// TIA Portal V19 export
FUNCTION "SET PARAMETER" : Void   // FC18, LAD
{ S7_Optimized_Access := 'TRUE' }
// stored: SetENOAutomatically false
   VAR_TEMP   // added for the SCL form of the ladder/FBD networks
      _w1 : Bool;
   END_VAR
BEGIN

REGION Network 1: MFG STIRRER MOTOR
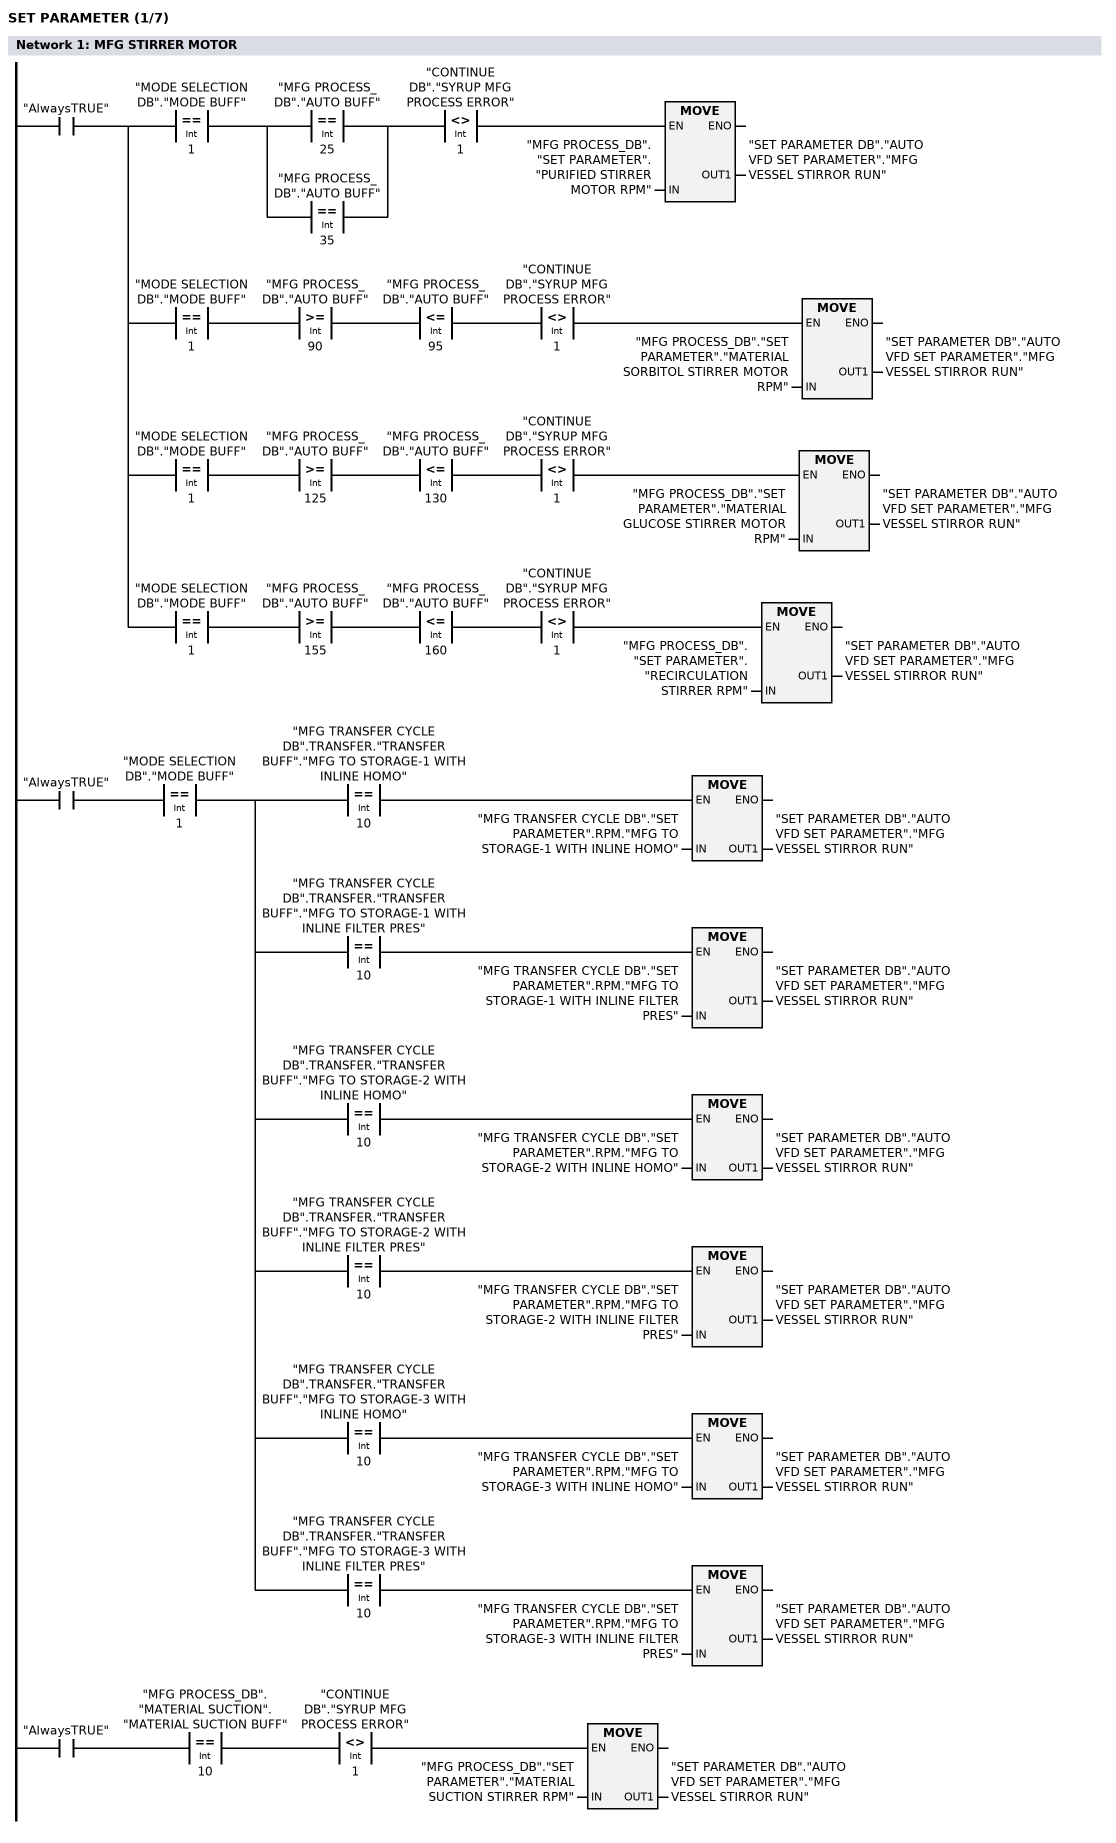
   RUNG wire#powerrail
      Contact( "AlwaysTRUE" )
      wire#w1
      { S7_Templates := "SrcType := Int" } EQ_Contact(in1 := "MODE SELECTION DB"."MODE BUFF", in2 := 1)
      wire#w2
      { S7_Templates := "SrcType := Int" } EQ_Contact(in1 := "MFG PROCESS_DB"."AUTO BUFF", in2 := 25)
      wire#w3
      { S7_Templates := "SrcType := Int" } NE_Contact(in1 := "CONTINUE DB"."SYRUP MFG PROCESS ERROR", in2 := 1)
      Move(in := "MFG PROCESS_DB"."SET PARAMETER"."PURIFIED STIRRER MOTOR RPM", out1 => "SET PARAMETER DB"."AUTO VFD SET PARAMETER"."MFG VESSEL STIRROR RUN")
   END_RUNG
   RUNG wire#w2
      { S7_Templates := "SrcType := Int" } EQ_Contact(in1 := "MFG PROCESS_DB"."AUTO BUFF", in2 := 35)
   END_RUNG wire#w3
   RUNG wire#w1
      { S7_Templates := "SrcType := Int" } EQ_Contact(in1 := "MODE SELECTION DB"."MODE BUFF", in2 := 1)
      { S7_Templates := "SrcType := Int" } GE_Contact(in1 := "MFG PROCESS_DB"."AUTO BUFF", in2 := 90)
      { S7_Templates := "SrcType := Int" } LE_Contact(in1 := "MFG PROCESS_DB"."AUTO BUFF", in2 := 95)
      { S7_Templates := "SrcType := Int" } NE_Contact(in1 := "CONTINUE DB"."SYRUP MFG PROCESS ERROR", in2 := 1)
      Move(in := "MFG PROCESS_DB"."SET PARAMETER"."MATERIAL SORBITOL STIRRER MOTOR RPM", out1 => "SET PARAMETER DB"."AUTO VFD SET PARAMETER"."MFG VESSEL STIRROR RUN")
   END_RUNG
   RUNG wire#w1
      { S7_Templates := "SrcType := Int" } EQ_Contact(in1 := "MODE SELECTION DB"."MODE BUFF", in2 := 1)
      { S7_Templates := "SrcType := Int" } GE_Contact(in1 := "MFG PROCESS_DB"."AUTO BUFF", in2 := 125)
      { S7_Templates := "SrcType := Int" } LE_Contact(in1 := "MFG PROCESS_DB"."AUTO BUFF", in2 := 130)
      { S7_Templates := "SrcType := Int" } NE_Contact(in1 := "CONTINUE DB"."SYRUP MFG PROCESS ERROR", in2 := 1)
      Move(in := "MFG PROCESS_DB"."SET PARAMETER"."MATERIAL GLUCOSE STIRRER MOTOR RPM", out1 => "SET PARAMETER DB"."AUTO VFD SET PARAMETER"."MFG VESSEL STIRROR RUN")
   END_RUNG
   RUNG wire#w1
      { S7_Templates := "SrcType := Int" } EQ_Contact(in1 := "MODE SELECTION DB"."MODE BUFF", in2 := 1)
      { S7_Templates := "SrcType := Int" } GE_Contact(in1 := "MFG PROCESS_DB"."AUTO BUFF", in2 := 155)
      { S7_Templates := "SrcType := Int" } LE_Contact(in1 := "MFG PROCESS_DB"."AUTO BUFF", in2 := 160)
      { S7_Templates := "SrcType := Int" } NE_Contact(in1 := "CONTINUE DB"."SYRUP MFG PROCESS ERROR", in2 := 1)
      Move(in := "MFG PROCESS_DB"."SET PARAMETER"."RECIRCULATION STIRRER RPM", out1 => "SET PARAMETER DB"."AUTO VFD SET PARAMETER"."MFG VESSEL STIRROR RUN")
   END_RUNG
   RUNG wire#powerrail
      Contact( "AlwaysTRUE" )
      { S7_Templates := "SrcType := Int" } EQ_Contact(in1 := "MODE SELECTION DB"."MODE BUFF", in2 := 1)
      wire#w4
      { S7_Templates := "SrcType := Int" } EQ_Contact(in1 := "MFG TRANSFER CYCLE DB".TRANSFER."TRANSFER BUFF"."MFG TO STORAGE-1 WITH INLINE HOMO", in2 := 10)
      Move(in := "MFG TRANSFER CYCLE DB"."SET PARAMETER".RPM."MFG TO STORAGE-1 WITH INLINE HOMO", out1 => "SET PARAMETER DB"."AUTO VFD SET PARAMETER"."MFG VESSEL STIRROR RUN")
   END_RUNG
   RUNG wire#w4
      { S7_Templates := "SrcType := Int" } EQ_Contact(in1 := "MFG TRANSFER CYCLE DB".TRANSFER."TRANSFER BUFF"."MFG TO STORAGE-1 WITH INLINE FILTER PRES", in2 := 10)
      Move(in := "MFG TRANSFER CYCLE DB"."SET PARAMETER".RPM."MFG TO STORAGE-1 WITH INLINE FILTER PRES", out1 => "SET PARAMETER DB"."AUTO VFD SET PARAMETER"."MFG VESSEL STIRROR RUN")
   END_RUNG
   RUNG wire#w4
      { S7_Templates := "SrcType := Int" } EQ_Contact(in1 := "MFG TRANSFER CYCLE DB".TRANSFER."TRANSFER BUFF"."MFG TO STORAGE-2 WITH INLINE HOMO", in2 := 10)
      Move(in := "MFG TRANSFER CYCLE DB"."SET PARAMETER".RPM."MFG TO STORAGE-2 WITH INLINE HOMO", out1 => "SET PARAMETER DB"."AUTO VFD SET PARAMETER"."MFG VESSEL STIRROR RUN")
   END_RUNG
   RUNG wire#w4
      { S7_Templates := "SrcType := Int" } EQ_Contact(in1 := "MFG TRANSFER CYCLE DB".TRANSFER."TRANSFER BUFF"."MFG TO STORAGE-2 WITH INLINE FILTER PRES", in2 := 10)
      Move(in := "MFG TRANSFER CYCLE DB"."SET PARAMETER".RPM."MFG TO STORAGE-2 WITH INLINE FILTER PRES", out1 => "SET PARAMETER DB"."AUTO VFD SET PARAMETER"."MFG VESSEL STIRROR RUN")
   END_RUNG
   RUNG wire#w4
      { S7_Templates := "SrcType := Int" } EQ_Contact(in1 := "MFG TRANSFER CYCLE DB".TRANSFER."TRANSFER BUFF"."MFG TO STORAGE-3 WITH INLINE HOMO", in2 := 10)
      Move(in := "MFG TRANSFER CYCLE DB"."SET PARAMETER".RPM."MFG TO STORAGE-3 WITH INLINE HOMO", out1 => "SET PARAMETER DB"."AUTO VFD SET PARAMETER"."MFG VESSEL STIRROR RUN")
   END_RUNG
   RUNG wire#w4
      { S7_Templates := "SrcType := Int" } EQ_Contact(in1 := "MFG TRANSFER CYCLE DB".TRANSFER."TRANSFER BUFF"."MFG TO STORAGE-3 WITH INLINE FILTER PRES", in2 := 10)
      Move(in := "MFG TRANSFER CYCLE DB"."SET PARAMETER".RPM."MFG TO STORAGE-3 WITH INLINE FILTER PRES", out1 => "SET PARAMETER DB"."AUTO VFD SET PARAMETER"."MFG VESSEL STIRROR RUN")
   END_RUNG
   RUNG wire#powerrail
      Contact( "AlwaysTRUE" )
      { S7_Templates := "SrcType := Int" } EQ_Contact(in1 := "MFG PROCESS_DB"."MATERIAL SUCTION"."MATERIAL SUCTION BUFF", in2 := 10)
      { S7_Templates := "SrcType := Int" } NE_Contact(in1 := "CONTINUE DB"."SYRUP MFG PROCESS ERROR", in2 := 1)
      Move(in := "MFG PROCESS_DB"."SET PARAMETER"."MATERIAL SUCTION STIRRER RPM", out1 => "SET PARAMETER DB"."AUTO VFD SET PARAMETER"."MFG VESSEL STIRROR RUN")
   END_RUNG
   // the same network as SCL:
   IF "AlwaysTRUE" AND ("MODE SELECTION DB"."MODE BUFF" = 1) AND (("MFG PROCESS_DB"."AUTO BUFF" = 25) OR ("MFG PROCESS_DB"."AUTO BUFF" = 35)) AND ("CONTINUE DB"."SYRUP MFG PROCESS ERROR" <> 1) THEN
       "SET PARAMETER DB"."AUTO VFD SET PARAMETER"."MFG VESSEL STIRROR RUN" := "MFG PROCESS_DB"."SET PARAMETER"."PURIFIED STIRRER MOTOR RPM";
   END_IF;
   IF "AlwaysTRUE" AND ("MODE SELECTION DB"."MODE BUFF" = 1) AND ("MFG PROCESS_DB"."AUTO BUFF" >= 90) AND ("MFG PROCESS_DB"."AUTO BUFF" <= 95) AND ("CONTINUE DB"."SYRUP MFG PROCESS ERROR" <> 1) THEN
       "SET PARAMETER DB"."AUTO VFD SET PARAMETER"."MFG VESSEL STIRROR RUN" := "MFG PROCESS_DB"."SET PARAMETER"."MATERIAL SORBITOL STIRRER MOTOR RPM";
   END_IF;
   IF "AlwaysTRUE" AND ("MODE SELECTION DB"."MODE BUFF" = 1) AND ("MFG PROCESS_DB"."AUTO BUFF" >= 125) AND ("MFG PROCESS_DB"."AUTO BUFF" <= 130) AND ("CONTINUE DB"."SYRUP MFG PROCESS ERROR" <> 1) THEN
       "SET PARAMETER DB"."AUTO VFD SET PARAMETER"."MFG VESSEL STIRROR RUN" := "MFG PROCESS_DB"."SET PARAMETER"."MATERIAL GLUCOSE STIRRER MOTOR RPM";
   END_IF;
   IF "AlwaysTRUE" AND ("MODE SELECTION DB"."MODE BUFF" = 1) AND ("MFG PROCESS_DB"."AUTO BUFF" >= 155) AND ("MFG PROCESS_DB"."AUTO BUFF" <= 160) AND ("CONTINUE DB"."SYRUP MFG PROCESS ERROR" <> 1) THEN
       "SET PARAMETER DB"."AUTO VFD SET PARAMETER"."MFG VESSEL STIRROR RUN" := "MFG PROCESS_DB"."SET PARAMETER"."RECIRCULATION STIRRER RPM";
   END_IF;
   #_w1 := "AlwaysTRUE" AND ("MODE SELECTION DB"."MODE BUFF" = 1);
   IF #_w1 AND ("MFG TRANSFER CYCLE DB".TRANSFER."TRANSFER BUFF"."MFG TO STORAGE-1 WITH INLINE HOMO" = 10) THEN
       "SET PARAMETER DB"."AUTO VFD SET PARAMETER"."MFG VESSEL STIRROR RUN" := "MFG TRANSFER CYCLE DB"."SET PARAMETER".RPM."MFG TO STORAGE-1 WITH INLINE HOMO";
   END_IF;
   IF #_w1 AND ("MFG TRANSFER CYCLE DB".TRANSFER."TRANSFER BUFF"."MFG TO STORAGE-1 WITH INLINE FILTER PRES" = 10) THEN
       "SET PARAMETER DB"."AUTO VFD SET PARAMETER"."MFG VESSEL STIRROR RUN" := "MFG TRANSFER CYCLE DB"."SET PARAMETER".RPM."MFG TO STORAGE-1 WITH INLINE FILTER PRES";
   END_IF;
   IF #_w1 AND ("MFG TRANSFER CYCLE DB".TRANSFER."TRANSFER BUFF"."MFG TO STORAGE-2 WITH INLINE HOMO" = 10) THEN
       "SET PARAMETER DB"."AUTO VFD SET PARAMETER"."MFG VESSEL STIRROR RUN" := "MFG TRANSFER CYCLE DB"."SET PARAMETER".RPM."MFG TO STORAGE-2 WITH INLINE HOMO";
   END_IF;
   IF #_w1 AND ("MFG TRANSFER CYCLE DB".TRANSFER."TRANSFER BUFF"."MFG TO STORAGE-2 WITH INLINE FILTER PRES" = 10) THEN
       "SET PARAMETER DB"."AUTO VFD SET PARAMETER"."MFG VESSEL STIRROR RUN" := "MFG TRANSFER CYCLE DB"."SET PARAMETER".RPM."MFG TO STORAGE-2 WITH INLINE FILTER PRES";
   END_IF;
   IF #_w1 AND ("MFG TRANSFER CYCLE DB".TRANSFER."TRANSFER BUFF"."MFG TO STORAGE-3 WITH INLINE HOMO" = 10) THEN
       "SET PARAMETER DB"."AUTO VFD SET PARAMETER"."MFG VESSEL STIRROR RUN" := "MFG TRANSFER CYCLE DB"."SET PARAMETER".RPM."MFG TO STORAGE-3 WITH INLINE HOMO";
   END_IF;
   IF #_w1 AND ("MFG TRANSFER CYCLE DB".TRANSFER."TRANSFER BUFF"."MFG TO STORAGE-3 WITH INLINE FILTER PRES" = 10) THEN
       "SET PARAMETER DB"."AUTO VFD SET PARAMETER"."MFG VESSEL STIRROR RUN" := "MFG TRANSFER CYCLE DB"."SET PARAMETER".RPM."MFG TO STORAGE-3 WITH INLINE FILTER PRES";
   END_IF;
   IF "AlwaysTRUE" AND ("MFG PROCESS_DB"."MATERIAL SUCTION"."MATERIAL SUCTION BUFF" = 10) AND ("CONTINUE DB"."SYRUP MFG PROCESS ERROR" <> 1) THEN
       "SET PARAMETER DB"."AUTO VFD SET PARAMETER"."MFG VESSEL STIRROR RUN" := "MFG PROCESS_DB"."SET PARAMETER"."MATERIAL SUCTION STIRRER RPM";
   END_IF;
END_REGION

REGION Network 2: PREMIXING STIRRER MOTOR
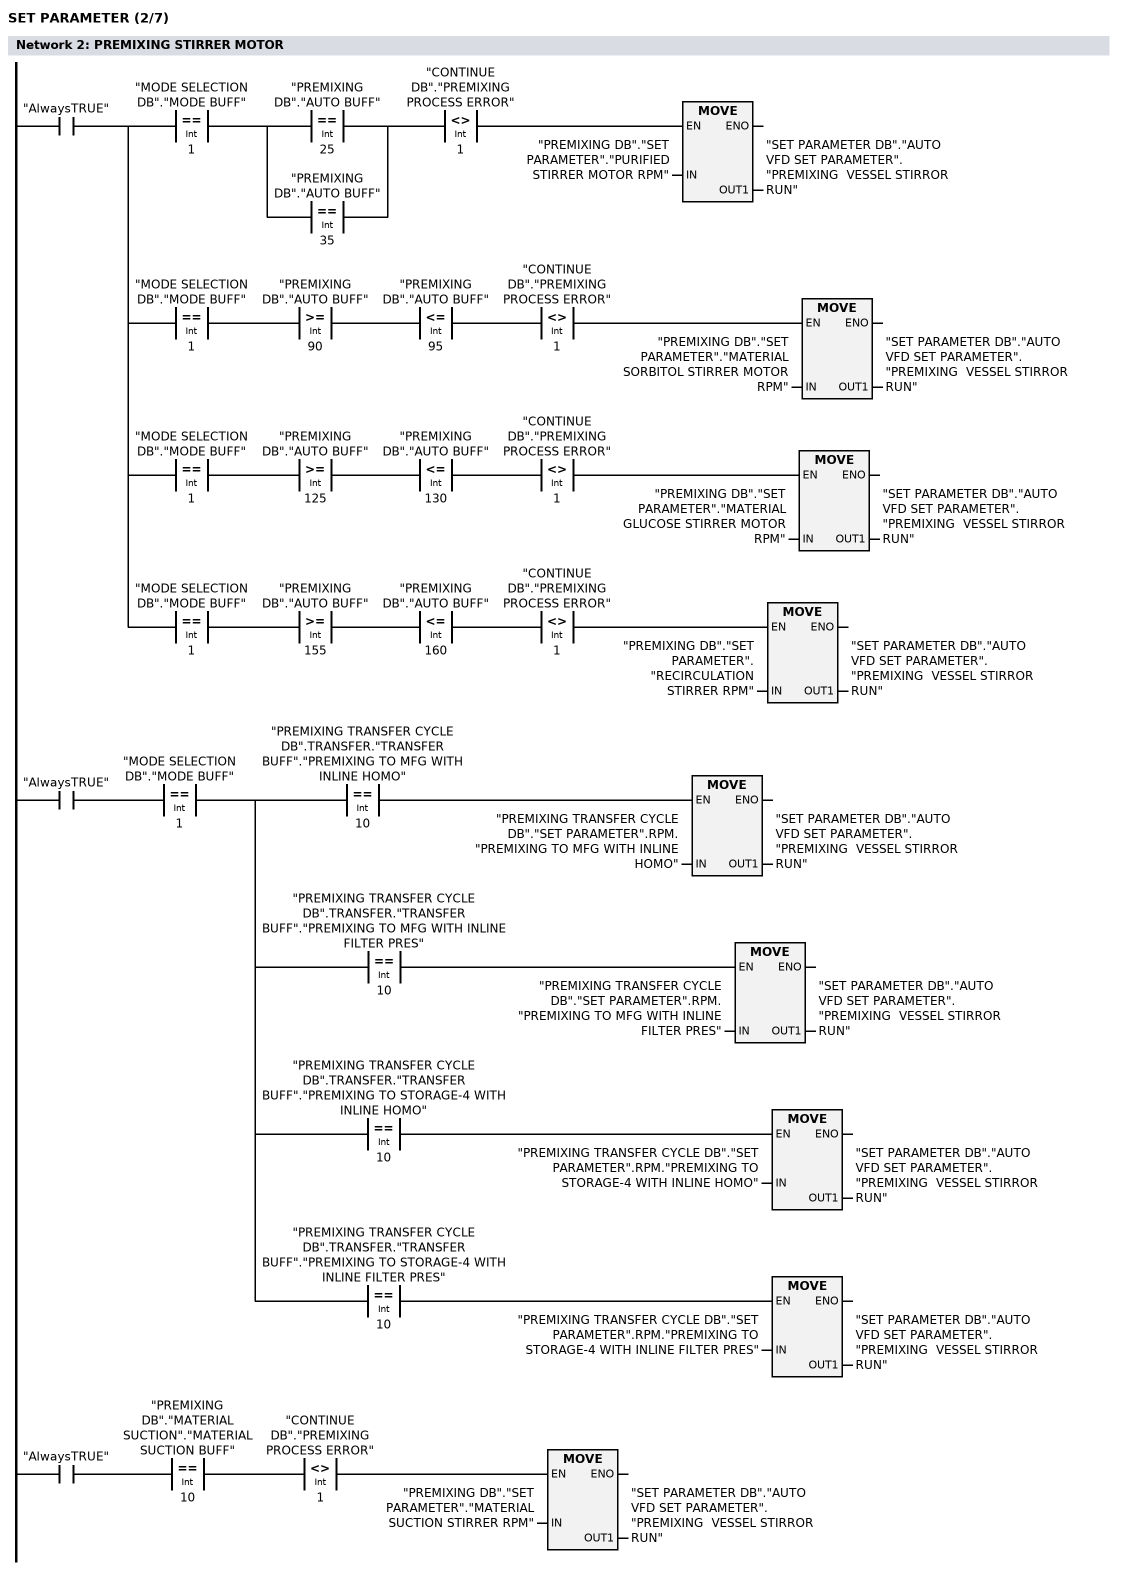
   RUNG wire#powerrail
      Contact( "AlwaysTRUE" )
      wire#w1
      { S7_Templates := "SrcType := Int" } EQ_Contact(in1 := "MODE SELECTION DB"."MODE BUFF", in2 := 1)
      wire#w2
      { S7_Templates := "SrcType := Int" } EQ_Contact(in1 := "PREMIXING DB"."AUTO BUFF", in2 := 25)
      wire#w3
      { S7_Templates := "SrcType := Int" } NE_Contact(in1 := "CONTINUE DB"."PREMIXING PROCESS ERROR", in2 := 1)
      Move(in := "PREMIXING DB"."SET PARAMETER"."PURIFIED STIRRER MOTOR RPM", out1 => "SET PARAMETER DB"."AUTO VFD SET PARAMETER"."PREMIXING  VESSEL STIRROR RUN")
   END_RUNG
   RUNG wire#w2
      { S7_Templates := "SrcType := Int" } EQ_Contact(in1 := "PREMIXING DB"."AUTO BUFF", in2 := 35)
   END_RUNG wire#w3
   RUNG wire#w1
      { S7_Templates := "SrcType := Int" } EQ_Contact(in1 := "MODE SELECTION DB"."MODE BUFF", in2 := 1)
      { S7_Templates := "SrcType := Int" } GE_Contact(in1 := "PREMIXING DB"."AUTO BUFF", in2 := 90)
      { S7_Templates := "SrcType := Int" } LE_Contact(in1 := "PREMIXING DB"."AUTO BUFF", in2 := 95)
      { S7_Templates := "SrcType := Int" } NE_Contact(in1 := "CONTINUE DB"."PREMIXING PROCESS ERROR", in2 := 1)
      Move(in := "PREMIXING DB"."SET PARAMETER"."MATERIAL SORBITOL STIRRER MOTOR RPM", out1 => "SET PARAMETER DB"."AUTO VFD SET PARAMETER"."PREMIXING  VESSEL STIRROR RUN")
   END_RUNG
   RUNG wire#w1
      { S7_Templates := "SrcType := Int" } EQ_Contact(in1 := "MODE SELECTION DB"."MODE BUFF", in2 := 1)
      { S7_Templates := "SrcType := Int" } GE_Contact(in1 := "PREMIXING DB"."AUTO BUFF", in2 := 125)
      { S7_Templates := "SrcType := Int" } LE_Contact(in1 := "PREMIXING DB"."AUTO BUFF", in2 := 130)
      { S7_Templates := "SrcType := Int" } NE_Contact(in1 := "CONTINUE DB"."PREMIXING PROCESS ERROR", in2 := 1)
      Move(in := "PREMIXING DB"."SET PARAMETER"."MATERIAL GLUCOSE STIRRER MOTOR RPM", out1 => "SET PARAMETER DB"."AUTO VFD SET PARAMETER"."PREMIXING  VESSEL STIRROR RUN")
   END_RUNG
   RUNG wire#w1
      { S7_Templates := "SrcType := Int" } EQ_Contact(in1 := "MODE SELECTION DB"."MODE BUFF", in2 := 1)
      { S7_Templates := "SrcType := Int" } GE_Contact(in1 := "PREMIXING DB"."AUTO BUFF", in2 := 155)
      { S7_Templates := "SrcType := Int" } LE_Contact(in1 := "PREMIXING DB"."AUTO BUFF", in2 := 160)
      { S7_Templates := "SrcType := Int" } NE_Contact(in1 := "CONTINUE DB"."PREMIXING PROCESS ERROR", in2 := 1)
      Move(in := "PREMIXING DB"."SET PARAMETER"."RECIRCULATION STIRRER RPM", out1 => "SET PARAMETER DB"."AUTO VFD SET PARAMETER"."PREMIXING  VESSEL STIRROR RUN")
   END_RUNG
   RUNG wire#powerrail
      Contact( "AlwaysTRUE" )
      { S7_Templates := "SrcType := Int" } EQ_Contact(in1 := "MODE SELECTION DB"."MODE BUFF", in2 := 1)
      wire#w4
      { S7_Templates := "SrcType := Int" } EQ_Contact(in1 := "PREMIXING TRANSFER CYCLE DB".TRANSFER."TRANSFER BUFF"."PREMIXING TO MFG WITH INLINE HOMO", in2 := 10)
      Move(in := "PREMIXING TRANSFER CYCLE DB"."SET PARAMETER".RPM."PREMIXING TO MFG WITH INLINE HOMO", out1 => "SET PARAMETER DB"."AUTO VFD SET PARAMETER"."PREMIXING  VESSEL STIRROR RUN")
   END_RUNG
   RUNG wire#w4
      { S7_Templates := "SrcType := Int" } EQ_Contact(in1 := "PREMIXING TRANSFER CYCLE DB".TRANSFER."TRANSFER BUFF"."PREMIXING TO MFG WITH INLINE FILTER PRES", in2 := 10)
      Move(in := "PREMIXING TRANSFER CYCLE DB"."SET PARAMETER".RPM."PREMIXING TO MFG WITH INLINE FILTER PRES", out1 => "SET PARAMETER DB"."AUTO VFD SET PARAMETER"."PREMIXING  VESSEL STIRROR RUN")
   END_RUNG
   RUNG wire#w4
      { S7_Templates := "SrcType := Int" } EQ_Contact(in1 := "PREMIXING TRANSFER CYCLE DB".TRANSFER."TRANSFER BUFF"."PREMIXING TO STORAGE-4 WITH INLINE HOMO", in2 := 10)
      Move(in := "PREMIXING TRANSFER CYCLE DB"."SET PARAMETER".RPM."PREMIXING TO STORAGE-4 WITH INLINE HOMO", out1 => "SET PARAMETER DB"."AUTO VFD SET PARAMETER"."PREMIXING  VESSEL STIRROR RUN")
   END_RUNG
   RUNG wire#w4
      { S7_Templates := "SrcType := Int" } EQ_Contact(in1 := "PREMIXING TRANSFER CYCLE DB".TRANSFER."TRANSFER BUFF"."PREMIXING TO STORAGE-4 WITH INLINE FILTER PRES", in2 := 10)
      Move(in := "PREMIXING TRANSFER CYCLE DB"."SET PARAMETER".RPM."PREMIXING TO STORAGE-4 WITH INLINE FILTER PRES", out1 => "SET PARAMETER DB"."AUTO VFD SET PARAMETER"."PREMIXING  VESSEL STIRROR RUN")
   END_RUNG
   RUNG wire#powerrail
      Contact( "AlwaysTRUE" )
      { S7_Templates := "SrcType := Int" } EQ_Contact(in1 := "PREMIXING DB"."MATERIAL SUCTION"."MATERIAL SUCTION BUFF", in2 := 10)
      { S7_Templates := "SrcType := Int" } NE_Contact(in1 := "CONTINUE DB"."PREMIXING PROCESS ERROR", in2 := 1)
      Move(in := "PREMIXING DB"."SET PARAMETER"."MATERIAL SUCTION STIRRER RPM", out1 => "SET PARAMETER DB"."AUTO VFD SET PARAMETER"."PREMIXING  VESSEL STIRROR RUN")
   END_RUNG
   // the same network as SCL:
   IF "AlwaysTRUE" AND ("MODE SELECTION DB"."MODE BUFF" = 1) AND (("PREMIXING DB"."AUTO BUFF" = 25) OR ("PREMIXING DB"."AUTO BUFF" = 35)) AND ("CONTINUE DB"."PREMIXING PROCESS ERROR" <> 1) THEN
       "SET PARAMETER DB"."AUTO VFD SET PARAMETER"."PREMIXING  VESSEL STIRROR RUN" := "PREMIXING DB"."SET PARAMETER"."PURIFIED STIRRER MOTOR RPM";
   END_IF;
   IF "AlwaysTRUE" AND ("MODE SELECTION DB"."MODE BUFF" = 1) AND ("PREMIXING DB"."AUTO BUFF" >= 90) AND ("PREMIXING DB"."AUTO BUFF" <= 95) AND ("CONTINUE DB"."PREMIXING PROCESS ERROR" <> 1) THEN
       "SET PARAMETER DB"."AUTO VFD SET PARAMETER"."PREMIXING  VESSEL STIRROR RUN" := "PREMIXING DB"."SET PARAMETER"."MATERIAL SORBITOL STIRRER MOTOR RPM";
   END_IF;
   IF "AlwaysTRUE" AND ("MODE SELECTION DB"."MODE BUFF" = 1) AND ("PREMIXING DB"."AUTO BUFF" >= 125) AND ("PREMIXING DB"."AUTO BUFF" <= 130) AND ("CONTINUE DB"."PREMIXING PROCESS ERROR" <> 1) THEN
       "SET PARAMETER DB"."AUTO VFD SET PARAMETER"."PREMIXING  VESSEL STIRROR RUN" := "PREMIXING DB"."SET PARAMETER"."MATERIAL GLUCOSE STIRRER MOTOR RPM";
   END_IF;
   IF "AlwaysTRUE" AND ("MODE SELECTION DB"."MODE BUFF" = 1) AND ("PREMIXING DB"."AUTO BUFF" >= 155) AND ("PREMIXING DB"."AUTO BUFF" <= 160) AND ("CONTINUE DB"."PREMIXING PROCESS ERROR" <> 1) THEN
       "SET PARAMETER DB"."AUTO VFD SET PARAMETER"."PREMIXING  VESSEL STIRROR RUN" := "PREMIXING DB"."SET PARAMETER"."RECIRCULATION STIRRER RPM";
   END_IF;
   #_w1 := "AlwaysTRUE" AND ("MODE SELECTION DB"."MODE BUFF" = 1);
   IF #_w1 AND ("PREMIXING TRANSFER CYCLE DB".TRANSFER."TRANSFER BUFF"."PREMIXING TO MFG WITH INLINE HOMO" = 10) THEN
       "SET PARAMETER DB"."AUTO VFD SET PARAMETER"."PREMIXING  VESSEL STIRROR RUN" := "PREMIXING TRANSFER CYCLE DB"."SET PARAMETER".RPM."PREMIXING TO MFG WITH INLINE HOMO";
   END_IF;
   IF #_w1 AND ("PREMIXING TRANSFER CYCLE DB".TRANSFER."TRANSFER BUFF"."PREMIXING TO MFG WITH INLINE FILTER PRES" = 10) THEN
       "SET PARAMETER DB"."AUTO VFD SET PARAMETER"."PREMIXING  VESSEL STIRROR RUN" := "PREMIXING TRANSFER CYCLE DB"."SET PARAMETER".RPM."PREMIXING TO MFG WITH INLINE FILTER PRES";
   END_IF;
   IF #_w1 AND ("PREMIXING TRANSFER CYCLE DB".TRANSFER."TRANSFER BUFF"."PREMIXING TO STORAGE-4 WITH INLINE HOMO" = 10) THEN
       "SET PARAMETER DB"."AUTO VFD SET PARAMETER"."PREMIXING  VESSEL STIRROR RUN" := "PREMIXING TRANSFER CYCLE DB"."SET PARAMETER".RPM."PREMIXING TO STORAGE-4 WITH INLINE HOMO";
   END_IF;
   IF #_w1 AND ("PREMIXING TRANSFER CYCLE DB".TRANSFER."TRANSFER BUFF"."PREMIXING TO STORAGE-4 WITH INLINE FILTER PRES" = 10) THEN
       "SET PARAMETER DB"."AUTO VFD SET PARAMETER"."PREMIXING  VESSEL STIRROR RUN" := "PREMIXING TRANSFER CYCLE DB"."SET PARAMETER".RPM."PREMIXING TO STORAGE-4 WITH INLINE FILTER PRES";
   END_IF;
   IF "AlwaysTRUE" AND ("PREMIXING DB"."MATERIAL SUCTION"."MATERIAL SUCTION BUFF" = 10) AND ("CONTINUE DB"."PREMIXING PROCESS ERROR" <> 1) THEN
       "SET PARAMETER DB"."AUTO VFD SET PARAMETER"."PREMIXING  VESSEL STIRROR RUN" := "PREMIXING DB"."SET PARAMETER"."MATERIAL SUCTION STIRRER RPM";
   END_IF;
END_REGION

REGION Network 3: SUGAR STIRRER MOTOR
END_REGION

REGION Network 5: MFG_TEMP
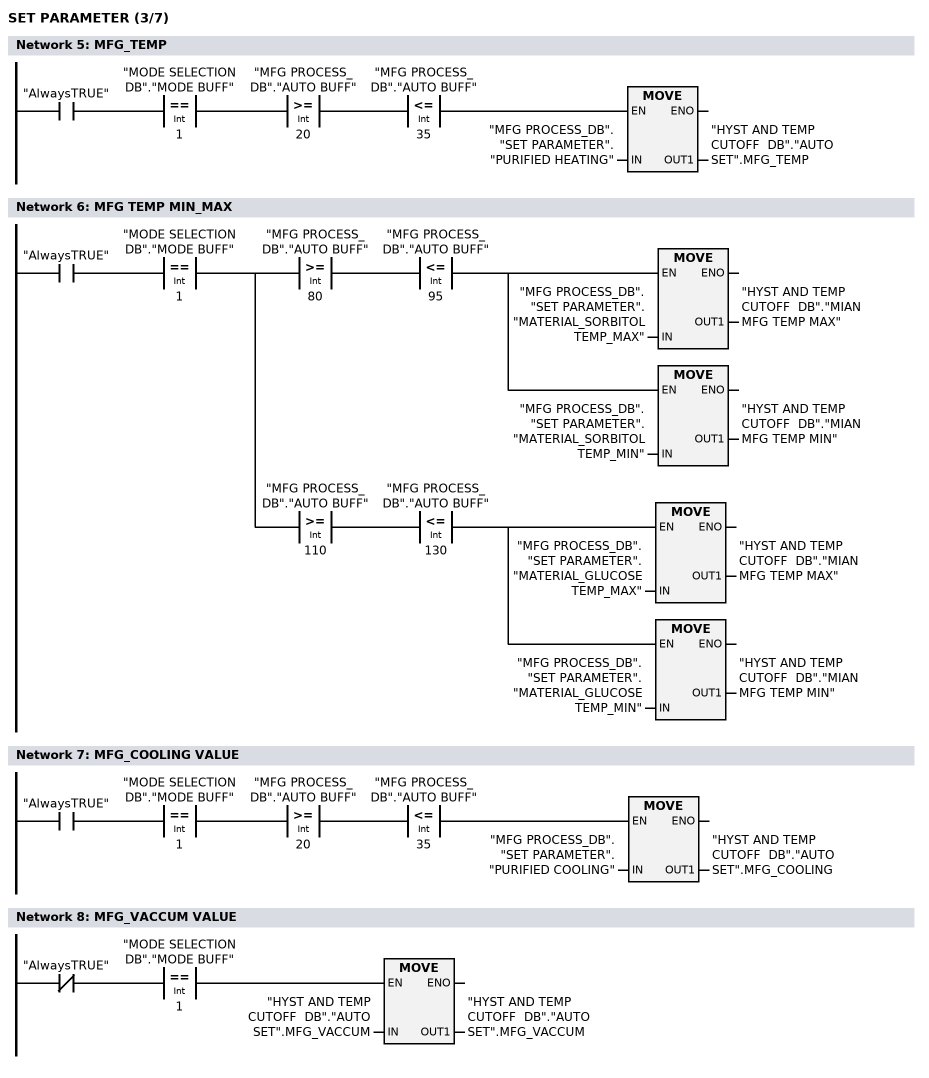
   RUNG wire#powerrail
      Contact( "AlwaysTRUE" )
      { S7_Templates := "SrcType := Int" } EQ_Contact(in1 := "MODE SELECTION DB"."MODE BUFF", in2 := 1)
      { S7_Templates := "SrcType := Int" } GE_Contact(in1 := "MFG PROCESS_DB"."AUTO BUFF", in2 := 20)
      { S7_Templates := "SrcType := Int" } LE_Contact(in1 := "MFG PROCESS_DB"."AUTO BUFF", in2 := 35)
      Move(in := "MFG PROCESS_DB"."SET PARAMETER"."PURIFIED HEATING", out1 => "HYST AND TEMP CUTOFF  DB"."AUTO SET".MFG_TEMP)
   END_RUNG
   // the same network as SCL:
   IF "AlwaysTRUE" AND ("MODE SELECTION DB"."MODE BUFF" = 1) AND ("MFG PROCESS_DB"."AUTO BUFF" >= 20) AND ("MFG PROCESS_DB"."AUTO BUFF" <= 35) THEN
       "HYST AND TEMP CUTOFF  DB"."AUTO SET".MFG_TEMP := "MFG PROCESS_DB"."SET PARAMETER"."PURIFIED HEATING";
   END_IF;
END_REGION

REGION Network 6: MFG TEMP MIN_MAX
   RUNG wire#powerrail
      Contact( "AlwaysTRUE" )
      { S7_Templates := "SrcType := Int" } EQ_Contact(in1 := "MODE SELECTION DB"."MODE BUFF", in2 := 1)
      wire#w1
      { S7_Templates := "SrcType := Int" } GE_Contact(in1 := "MFG PROCESS_DB"."AUTO BUFF", in2 := 80)
      { S7_Templates := "SrcType := Int" } LE_Contact(in1 := "MFG PROCESS_DB"."AUTO BUFF", in2 := 95)
      wire#w2
      Move(in := "MFG PROCESS_DB"."SET PARAMETER"."MATERIAL_SORBITOL TEMP_MAX", out1 => "HYST AND TEMP CUTOFF  DB"."MIAN MFG TEMP MAX")
   END_RUNG
   RUNG wire#w2
      Move(in := "MFG PROCESS_DB"."SET PARAMETER"."MATERIAL_SORBITOL TEMP_MIN", out1 => "HYST AND TEMP CUTOFF  DB"."MIAN MFG TEMP MIN")
   END_RUNG
   RUNG wire#w1
      { S7_Templates := "SrcType := Int" } GE_Contact(in1 := "MFG PROCESS_DB"."AUTO BUFF", in2 := 110)
      { S7_Templates := "SrcType := Int" } LE_Contact(in1 := "MFG PROCESS_DB"."AUTO BUFF", in2 := 130)
      wire#w3
      Move(in := "MFG PROCESS_DB"."SET PARAMETER"."MATERIAL_GLUCOSE TEMP_MAX", out1 => "HYST AND TEMP CUTOFF  DB"."MIAN MFG TEMP MAX")
   END_RUNG
   RUNG wire#w3
      Move(in := "MFG PROCESS_DB"."SET PARAMETER"."MATERIAL_GLUCOSE TEMP_MIN", out1 => "HYST AND TEMP CUTOFF  DB"."MIAN MFG TEMP MIN")
   END_RUNG
   // the same network as SCL:
   #_w1 := "AlwaysTRUE" AND ("MODE SELECTION DB"."MODE BUFF" = 1);
   IF #_w1 AND ("MFG PROCESS_DB"."AUTO BUFF" >= 80) AND ("MFG PROCESS_DB"."AUTO BUFF" <= 95) THEN
       "HYST AND TEMP CUTOFF  DB"."MIAN MFG TEMP MAX" := "MFG PROCESS_DB"."SET PARAMETER"."MATERIAL_SORBITOL TEMP_MAX";
       "HYST AND TEMP CUTOFF  DB"."MIAN MFG TEMP MIN" := "MFG PROCESS_DB"."SET PARAMETER"."MATERIAL_SORBITOL TEMP_MIN";
   END_IF;
   IF #_w1 AND ("MFG PROCESS_DB"."AUTO BUFF" >= 110) AND ("MFG PROCESS_DB"."AUTO BUFF" <= 130) THEN
       "HYST AND TEMP CUTOFF  DB"."MIAN MFG TEMP MAX" := "MFG PROCESS_DB"."SET PARAMETER"."MATERIAL_GLUCOSE TEMP_MAX";
       "HYST AND TEMP CUTOFF  DB"."MIAN MFG TEMP MIN" := "MFG PROCESS_DB"."SET PARAMETER"."MATERIAL_GLUCOSE TEMP_MIN";
   END_IF;
END_REGION

REGION Network 7: MFG_COOLING VALUE
   RUNG wire#powerrail
      Contact( "AlwaysTRUE" )
      { S7_Templates := "SrcType := Int" } EQ_Contact(in1 := "MODE SELECTION DB"."MODE BUFF", in2 := 1)
      { S7_Templates := "SrcType := Int" } GE_Contact(in1 := "MFG PROCESS_DB"."AUTO BUFF", in2 := 20)
      { S7_Templates := "SrcType := Int" } LE_Contact(in1 := "MFG PROCESS_DB"."AUTO BUFF", in2 := 35)
      Move(in := "MFG PROCESS_DB"."SET PARAMETER"."PURIFIED COOLING", out1 => "HYST AND TEMP CUTOFF  DB"."AUTO SET".MFG_COOLING)
   END_RUNG
   // the same network as SCL:
   IF "AlwaysTRUE" AND ("MODE SELECTION DB"."MODE BUFF" = 1) AND ("MFG PROCESS_DB"."AUTO BUFF" >= 20) AND ("MFG PROCESS_DB"."AUTO BUFF" <= 35) THEN
       "HYST AND TEMP CUTOFF  DB"."AUTO SET".MFG_COOLING := "MFG PROCESS_DB"."SET PARAMETER"."PURIFIED COOLING";
   END_IF;
END_REGION

REGION Network 8: MFG_VACCUM VALUE
   RUNG wire#powerrail
      I_Contact( "AlwaysTRUE" )
      { S7_Templates := "SrcType := Int" } EQ_Contact(in1 := "MODE SELECTION DB"."MODE BUFF", in2 := 1)
      Move(in := "HYST AND TEMP CUTOFF  DB"."AUTO SET".MFG_VACCUM, out1 => "HYST AND TEMP CUTOFF  DB"."AUTO SET".MFG_VACCUM)
   END_RUNG
   // the same network as SCL:
   IF NOT "AlwaysTRUE" AND ("MODE SELECTION DB"."MODE BUFF" = 1) THEN
       "HYST AND TEMP CUTOFF  DB"."AUTO SET".MFG_VACCUM := "HYST AND TEMP CUTOFF  DB"."AUTO SET".MFG_VACCUM;
   END_IF;
END_REGION

REGION Network 9: AUTO MFG LOAD CELL FOR TRANSFER
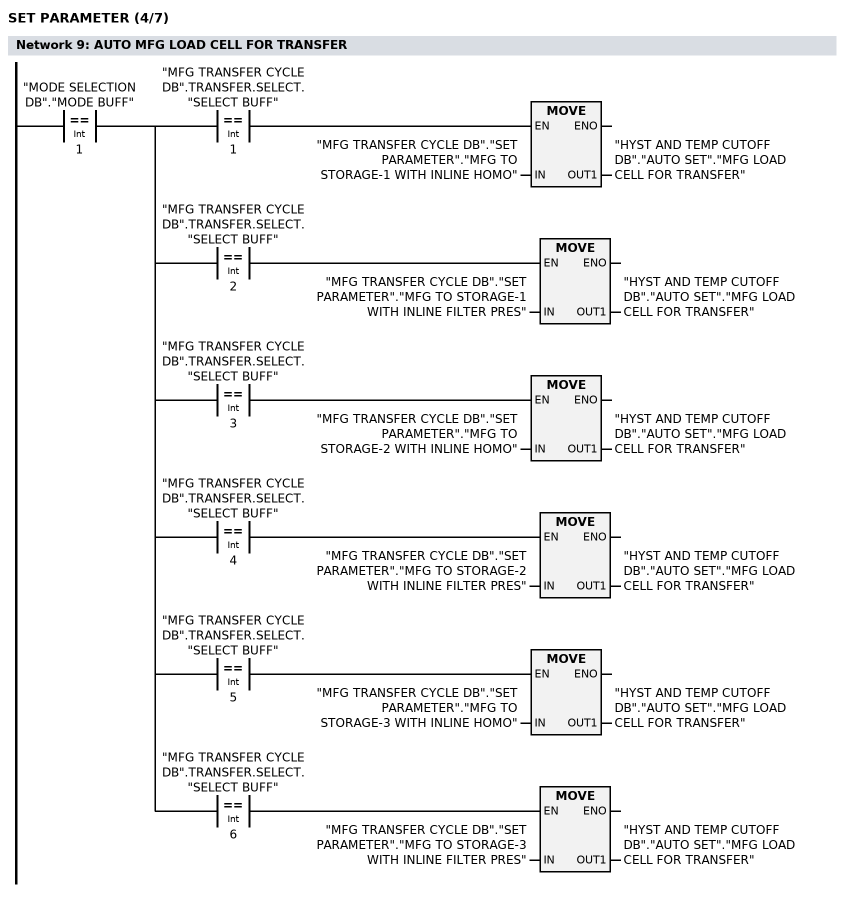
   RUNG wire#powerrail
      { S7_Templates := "SrcType := Int" } EQ_Contact(in1 := "MODE SELECTION DB"."MODE BUFF", in2 := 1)
      wire#w1
      { S7_Templates := "SrcType := Int" } EQ_Contact(in1 := "MFG TRANSFER CYCLE DB".TRANSFER.SELECT."SELECT BUFF", in2 := 1)
      Move(in := "MFG TRANSFER CYCLE DB"."SET PARAMETER"."MFG TO STORAGE-1 WITH INLINE HOMO", out1 => "HYST AND TEMP CUTOFF  DB"."AUTO SET"."MFG LOAD CELL FOR TRANSFER")
   END_RUNG
   RUNG wire#w1
      { S7_Templates := "SrcType := Int" } EQ_Contact(in1 := "MFG TRANSFER CYCLE DB".TRANSFER.SELECT."SELECT BUFF", in2 := 2)
      Move(in := "MFG TRANSFER CYCLE DB"."SET PARAMETER"."MFG TO STORAGE-1 WITH INLINE FILTER PRES", out1 => "HYST AND TEMP CUTOFF  DB"."AUTO SET"."MFG LOAD CELL FOR TRANSFER")
   END_RUNG
   RUNG wire#w1
      { S7_Templates := "SrcType := Int" } EQ_Contact(in1 := "MFG TRANSFER CYCLE DB".TRANSFER.SELECT."SELECT BUFF", in2 := 3)
      Move(in := "MFG TRANSFER CYCLE DB"."SET PARAMETER"."MFG TO STORAGE-2 WITH INLINE HOMO", out1 => "HYST AND TEMP CUTOFF  DB"."AUTO SET"."MFG LOAD CELL FOR TRANSFER")
   END_RUNG
   RUNG wire#w1
      { S7_Templates := "SrcType := Int" } EQ_Contact(in1 := "MFG TRANSFER CYCLE DB".TRANSFER.SELECT."SELECT BUFF", in2 := 4)
      Move(in := "MFG TRANSFER CYCLE DB"."SET PARAMETER"."MFG TO STORAGE-2 WITH INLINE FILTER PRES", out1 => "HYST AND TEMP CUTOFF  DB"."AUTO SET"."MFG LOAD CELL FOR TRANSFER")
   END_RUNG
   RUNG wire#w1
      { S7_Templates := "SrcType := Int" } EQ_Contact(in1 := "MFG TRANSFER CYCLE DB".TRANSFER.SELECT."SELECT BUFF", in2 := 5)
      Move(in := "MFG TRANSFER CYCLE DB"."SET PARAMETER"."MFG TO STORAGE-3 WITH INLINE HOMO", out1 => "HYST AND TEMP CUTOFF  DB"."AUTO SET"."MFG LOAD CELL FOR TRANSFER")
   END_RUNG
   RUNG wire#w1
      { S7_Templates := "SrcType := Int" } EQ_Contact(in1 := "MFG TRANSFER CYCLE DB".TRANSFER.SELECT."SELECT BUFF", in2 := 6)
      Move(in := "MFG TRANSFER CYCLE DB"."SET PARAMETER"."MFG TO STORAGE-3 WITH INLINE FILTER PRES", out1 => "HYST AND TEMP CUTOFF  DB"."AUTO SET"."MFG LOAD CELL FOR TRANSFER")
   END_RUNG
   // the same network as SCL:
   #_w1 := "MODE SELECTION DB"."MODE BUFF" = 1;
   IF #_w1 AND ("MFG TRANSFER CYCLE DB".TRANSFER.SELECT."SELECT BUFF" = 1) THEN
       "HYST AND TEMP CUTOFF  DB"."AUTO SET"."MFG LOAD CELL FOR TRANSFER" := "MFG TRANSFER CYCLE DB"."SET PARAMETER"."MFG TO STORAGE-1 WITH INLINE HOMO";
   END_IF;
   IF #_w1 AND ("MFG TRANSFER CYCLE DB".TRANSFER.SELECT."SELECT BUFF" = 2) THEN
       "HYST AND TEMP CUTOFF  DB"."AUTO SET"."MFG LOAD CELL FOR TRANSFER" := "MFG TRANSFER CYCLE DB"."SET PARAMETER"."MFG TO STORAGE-1 WITH INLINE FILTER PRES";
   END_IF;
   IF #_w1 AND ("MFG TRANSFER CYCLE DB".TRANSFER.SELECT."SELECT BUFF" = 3) THEN
       "HYST AND TEMP CUTOFF  DB"."AUTO SET"."MFG LOAD CELL FOR TRANSFER" := "MFG TRANSFER CYCLE DB"."SET PARAMETER"."MFG TO STORAGE-2 WITH INLINE HOMO";
   END_IF;
   IF #_w1 AND ("MFG TRANSFER CYCLE DB".TRANSFER.SELECT."SELECT BUFF" = 4) THEN
       "HYST AND TEMP CUTOFF  DB"."AUTO SET"."MFG LOAD CELL FOR TRANSFER" := "MFG TRANSFER CYCLE DB"."SET PARAMETER"."MFG TO STORAGE-2 WITH INLINE FILTER PRES";
   END_IF;
   IF #_w1 AND ("MFG TRANSFER CYCLE DB".TRANSFER.SELECT."SELECT BUFF" = 5) THEN
       "HYST AND TEMP CUTOFF  DB"."AUTO SET"."MFG LOAD CELL FOR TRANSFER" := "MFG TRANSFER CYCLE DB"."SET PARAMETER"."MFG TO STORAGE-3 WITH INLINE HOMO";
   END_IF;
   IF #_w1 AND ("MFG TRANSFER CYCLE DB".TRANSFER.SELECT."SELECT BUFF" = 6) THEN
       "HYST AND TEMP CUTOFF  DB"."AUTO SET"."MFG LOAD CELL FOR TRANSFER" := "MFG TRANSFER CYCLE DB"."SET PARAMETER"."MFG TO STORAGE-3 WITH INLINE FILTER PRES";
   END_IF;
END_REGION

REGION Network 10: AUTO MFG LOAD CELL VALUE
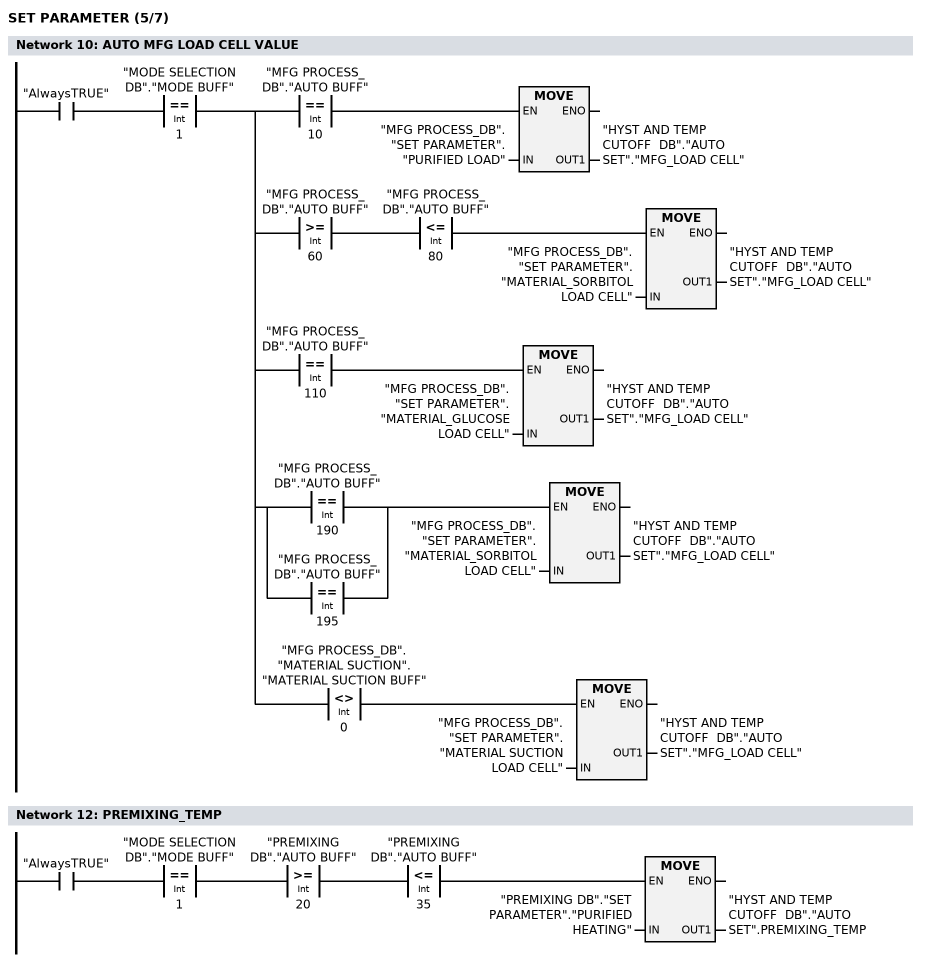
   RUNG wire#powerrail
      Contact( "AlwaysTRUE" )
      { S7_Templates := "SrcType := Int" } EQ_Contact(in1 := "MODE SELECTION DB"."MODE BUFF", in2 := 1)
      wire#w1
      { S7_Templates := "SrcType := Int" } EQ_Contact(in1 := "MFG PROCESS_DB"."AUTO BUFF", in2 := 10)
      Move(in := "MFG PROCESS_DB"."SET PARAMETER"."PURIFIED LOAD", out1 => "HYST AND TEMP CUTOFF  DB"."AUTO SET"."MFG_LOAD CELL")
   END_RUNG
   RUNG wire#w1
      { S7_Templates := "SrcType := Int" } GE_Contact(in1 := "MFG PROCESS_DB"."AUTO BUFF", in2 := 60)
      { S7_Templates := "SrcType := Int" } LE_Contact(in1 := "MFG PROCESS_DB"."AUTO BUFF", in2 := 80)
      Move(in := "MFG PROCESS_DB"."SET PARAMETER"."MATERIAL_SORBITOL LOAD CELL", out1 => "HYST AND TEMP CUTOFF  DB"."AUTO SET"."MFG_LOAD CELL")
   END_RUNG
   RUNG wire#w1
      { S7_Templates := "SrcType := Int" } EQ_Contact(in1 := "MFG PROCESS_DB"."AUTO BUFF", in2 := 110)
      Move(in := "MFG PROCESS_DB"."SET PARAMETER"."MATERIAL_GLUCOSE LOAD CELL", out1 => "HYST AND TEMP CUTOFF  DB"."AUTO SET"."MFG_LOAD CELL")
   END_RUNG
   RUNG wire#w1
      { S7_Templates := "SrcType := Int" } EQ_Contact(in1 := "MFG PROCESS_DB"."AUTO BUFF", in2 := 190)
      wire#w2
      Move(in := "MFG PROCESS_DB"."SET PARAMETER"."MATERIAL_SORBITOL LOAD CELL", out1 => "HYST AND TEMP CUTOFF  DB"."AUTO SET"."MFG_LOAD CELL")
   END_RUNG
   RUNG wire#w1
      { S7_Templates := "SrcType := Int" } EQ_Contact(in1 := "MFG PROCESS_DB"."AUTO BUFF", in2 := 195)
   END_RUNG wire#w2
   RUNG wire#w1
      { S7_Templates := "SrcType := Int" } NE_Contact(in1 := "MFG PROCESS_DB"."MATERIAL SUCTION"."MATERIAL SUCTION BUFF", in2 := 0)
      Move(in := "MFG PROCESS_DB"."SET PARAMETER"."MATERIAL SUCTION LOAD CELL", out1 => "HYST AND TEMP CUTOFF  DB"."AUTO SET"."MFG_LOAD CELL")
   END_RUNG
   // the same network as SCL:
   #_w1 := "AlwaysTRUE" AND ("MODE SELECTION DB"."MODE BUFF" = 1);
   IF #_w1 AND ("MFG PROCESS_DB"."AUTO BUFF" = 10) THEN
       "HYST AND TEMP CUTOFF  DB"."AUTO SET"."MFG_LOAD CELL" := "MFG PROCESS_DB"."SET PARAMETER"."PURIFIED LOAD";
   END_IF;
   IF #_w1 AND ("MFG PROCESS_DB"."AUTO BUFF" >= 60) AND ("MFG PROCESS_DB"."AUTO BUFF" <= 80) THEN
       "HYST AND TEMP CUTOFF  DB"."AUTO SET"."MFG_LOAD CELL" := "MFG PROCESS_DB"."SET PARAMETER"."MATERIAL_SORBITOL LOAD CELL";
   END_IF;
   IF #_w1 AND ("MFG PROCESS_DB"."AUTO BUFF" = 110) THEN
       "HYST AND TEMP CUTOFF  DB"."AUTO SET"."MFG_LOAD CELL" := "MFG PROCESS_DB"."SET PARAMETER"."MATERIAL_GLUCOSE LOAD CELL";
   END_IF;
   IF #_w1 AND (("MFG PROCESS_DB"."AUTO BUFF" = 190) OR ("MFG PROCESS_DB"."AUTO BUFF" = 195)) THEN
       "HYST AND TEMP CUTOFF  DB"."AUTO SET"."MFG_LOAD CELL" := "MFG PROCESS_DB"."SET PARAMETER"."MATERIAL_SORBITOL LOAD CELL";
   END_IF;
   IF #_w1 AND ("MFG PROCESS_DB"."MATERIAL SUCTION"."MATERIAL SUCTION BUFF" <> 0) THEN
       "HYST AND TEMP CUTOFF  DB"."AUTO SET"."MFG_LOAD CELL" := "MFG PROCESS_DB"."SET PARAMETER"."MATERIAL SUCTION LOAD CELL";
   END_IF;
END_REGION

REGION Network 12: PREMIXING_TEMP
   RUNG wire#powerrail
      Contact( "AlwaysTRUE" )
      { S7_Templates := "SrcType := Int" } EQ_Contact(in1 := "MODE SELECTION DB"."MODE BUFF", in2 := 1)
      { S7_Templates := "SrcType := Int" } GE_Contact(in1 := "PREMIXING DB"."AUTO BUFF", in2 := 20)
      { S7_Templates := "SrcType := Int" } LE_Contact(in1 := "PREMIXING DB"."AUTO BUFF", in2 := 35)
      Move(in := "PREMIXING DB"."SET PARAMETER"."PURIFIED HEATING", out1 => "HYST AND TEMP CUTOFF  DB"."AUTO SET".PREMIXING_TEMP)
   END_RUNG
   // the same network as SCL:
   IF "AlwaysTRUE" AND ("MODE SELECTION DB"."MODE BUFF" = 1) AND ("PREMIXING DB"."AUTO BUFF" >= 20) AND ("PREMIXING DB"."AUTO BUFF" <= 35) THEN
       "HYST AND TEMP CUTOFF  DB"."AUTO SET".PREMIXING_TEMP := "PREMIXING DB"."SET PARAMETER"."PURIFIED HEATING";
   END_IF;
END_REGION

REGION Network 13: PREMIXING TEMP MIN_MAX
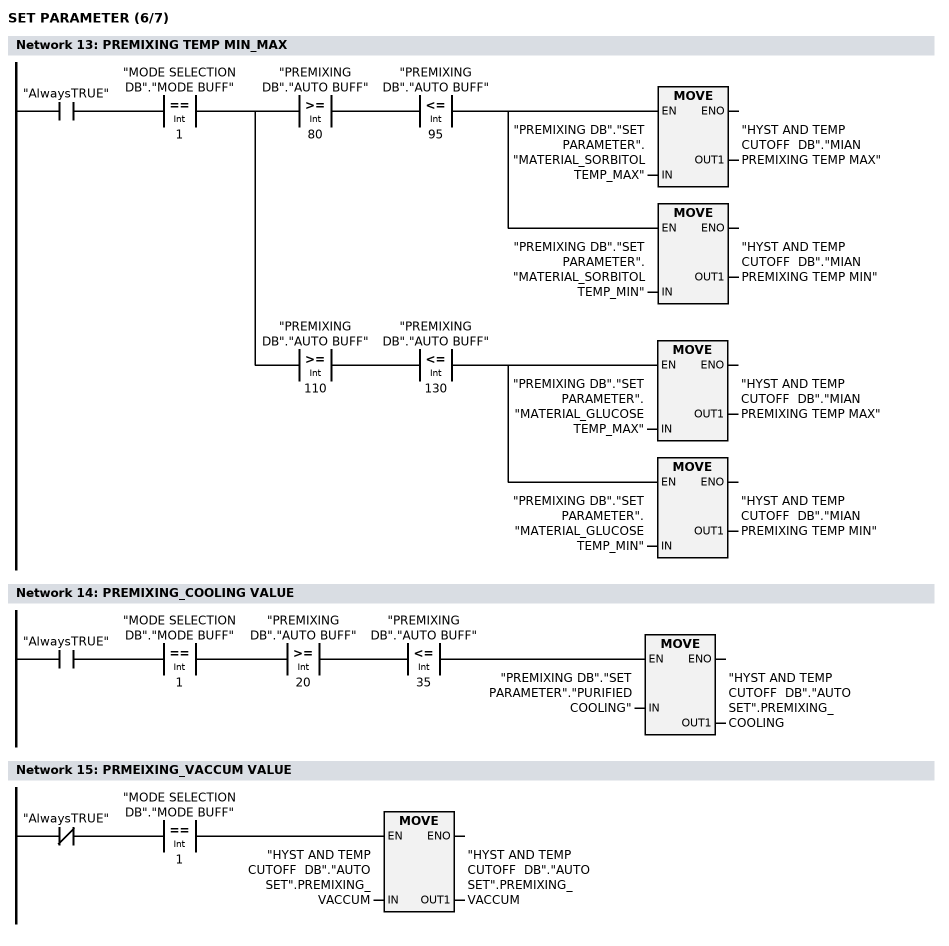
   RUNG wire#powerrail
      Contact( "AlwaysTRUE" )
      { S7_Templates := "SrcType := Int" } EQ_Contact(in1 := "MODE SELECTION DB"."MODE BUFF", in2 := 1)
      wire#w1
      { S7_Templates := "SrcType := Int" } GE_Contact(in1 := "PREMIXING DB"."AUTO BUFF", in2 := 80)
      { S7_Templates := "SrcType := Int" } LE_Contact(in1 := "PREMIXING DB"."AUTO BUFF", in2 := 95)
      wire#w2
      Move(in := "PREMIXING DB"."SET PARAMETER"."MATERIAL_SORBITOL TEMP_MAX", out1 => "HYST AND TEMP CUTOFF  DB"."MIAN PREMIXING TEMP MAX")
   END_RUNG
   RUNG wire#w2
      Move(in := "PREMIXING DB"."SET PARAMETER"."MATERIAL_SORBITOL TEMP_MIN", out1 => "HYST AND TEMP CUTOFF  DB"."MIAN PREMIXING TEMP MIN")
   END_RUNG
   RUNG wire#w1
      { S7_Templates := "SrcType := Int" } GE_Contact(in1 := "PREMIXING DB"."AUTO BUFF", in2 := 110)
      { S7_Templates := "SrcType := Int" } LE_Contact(in1 := "PREMIXING DB"."AUTO BUFF", in2 := 130)
      wire#w3
      Move(in := "PREMIXING DB"."SET PARAMETER"."MATERIAL_GLUCOSE TEMP_MAX", out1 => "HYST AND TEMP CUTOFF  DB"."MIAN PREMIXING TEMP MAX")
   END_RUNG
   RUNG wire#w3
      Move(in := "PREMIXING DB"."SET PARAMETER"."MATERIAL_GLUCOSE TEMP_MIN", out1 => "HYST AND TEMP CUTOFF  DB"."MIAN PREMIXING TEMP MIN")
   END_RUNG
   // the same network as SCL:
   #_w1 := "AlwaysTRUE" AND ("MODE SELECTION DB"."MODE BUFF" = 1);
   IF #_w1 AND ("PREMIXING DB"."AUTO BUFF" >= 80) AND ("PREMIXING DB"."AUTO BUFF" <= 95) THEN
       "HYST AND TEMP CUTOFF  DB"."MIAN PREMIXING TEMP MAX" := "PREMIXING DB"."SET PARAMETER"."MATERIAL_SORBITOL TEMP_MAX";
       "HYST AND TEMP CUTOFF  DB"."MIAN PREMIXING TEMP MIN" := "PREMIXING DB"."SET PARAMETER"."MATERIAL_SORBITOL TEMP_MIN";
   END_IF;
   IF #_w1 AND ("PREMIXING DB"."AUTO BUFF" >= 110) AND ("PREMIXING DB"."AUTO BUFF" <= 130) THEN
       "HYST AND TEMP CUTOFF  DB"."MIAN PREMIXING TEMP MAX" := "PREMIXING DB"."SET PARAMETER"."MATERIAL_GLUCOSE TEMP_MAX";
       "HYST AND TEMP CUTOFF  DB"."MIAN PREMIXING TEMP MIN" := "PREMIXING DB"."SET PARAMETER"."MATERIAL_GLUCOSE TEMP_MIN";
   END_IF;
END_REGION

REGION Network 14: PREMIXING_COOLING VALUE
   RUNG wire#powerrail
      Contact( "AlwaysTRUE" )
      { S7_Templates := "SrcType := Int" } EQ_Contact(in1 := "MODE SELECTION DB"."MODE BUFF", in2 := 1)
      { S7_Templates := "SrcType := Int" } GE_Contact(in1 := "PREMIXING DB"."AUTO BUFF", in2 := 20)
      { S7_Templates := "SrcType := Int" } LE_Contact(in1 := "PREMIXING DB"."AUTO BUFF", in2 := 35)
      Move(in := "PREMIXING DB"."SET PARAMETER"."PURIFIED COOLING", out1 => "HYST AND TEMP CUTOFF  DB"."AUTO SET".PREMIXING_COOLING)
   END_RUNG
   // the same network as SCL:
   IF "AlwaysTRUE" AND ("MODE SELECTION DB"."MODE BUFF" = 1) AND ("PREMIXING DB"."AUTO BUFF" >= 20) AND ("PREMIXING DB"."AUTO BUFF" <= 35) THEN
       "HYST AND TEMP CUTOFF  DB"."AUTO SET".PREMIXING_COOLING := "PREMIXING DB"."SET PARAMETER"."PURIFIED COOLING";
   END_IF;
END_REGION

REGION Network 15: PRMEIXING_VACCUM VALUE
   RUNG wire#powerrail
      I_Contact( "AlwaysTRUE" )
      { S7_Templates := "SrcType := Int" } EQ_Contact(in1 := "MODE SELECTION DB"."MODE BUFF", in2 := 1)
      Move(in := "HYST AND TEMP CUTOFF  DB"."AUTO SET".PREMIXING_VACCUM, out1 => "HYST AND TEMP CUTOFF  DB"."AUTO SET".PREMIXING_VACCUM)
   END_RUNG
   // the same network as SCL:
   IF NOT "AlwaysTRUE" AND ("MODE SELECTION DB"."MODE BUFF" = 1) THEN
       "HYST AND TEMP CUTOFF  DB"."AUTO SET".PREMIXING_VACCUM := "HYST AND TEMP CUTOFF  DB"."AUTO SET".PREMIXING_VACCUM;
   END_IF;
END_REGION

REGION Network 16: AUTO PREMIXING LOAD CELL FOR TRANSFER
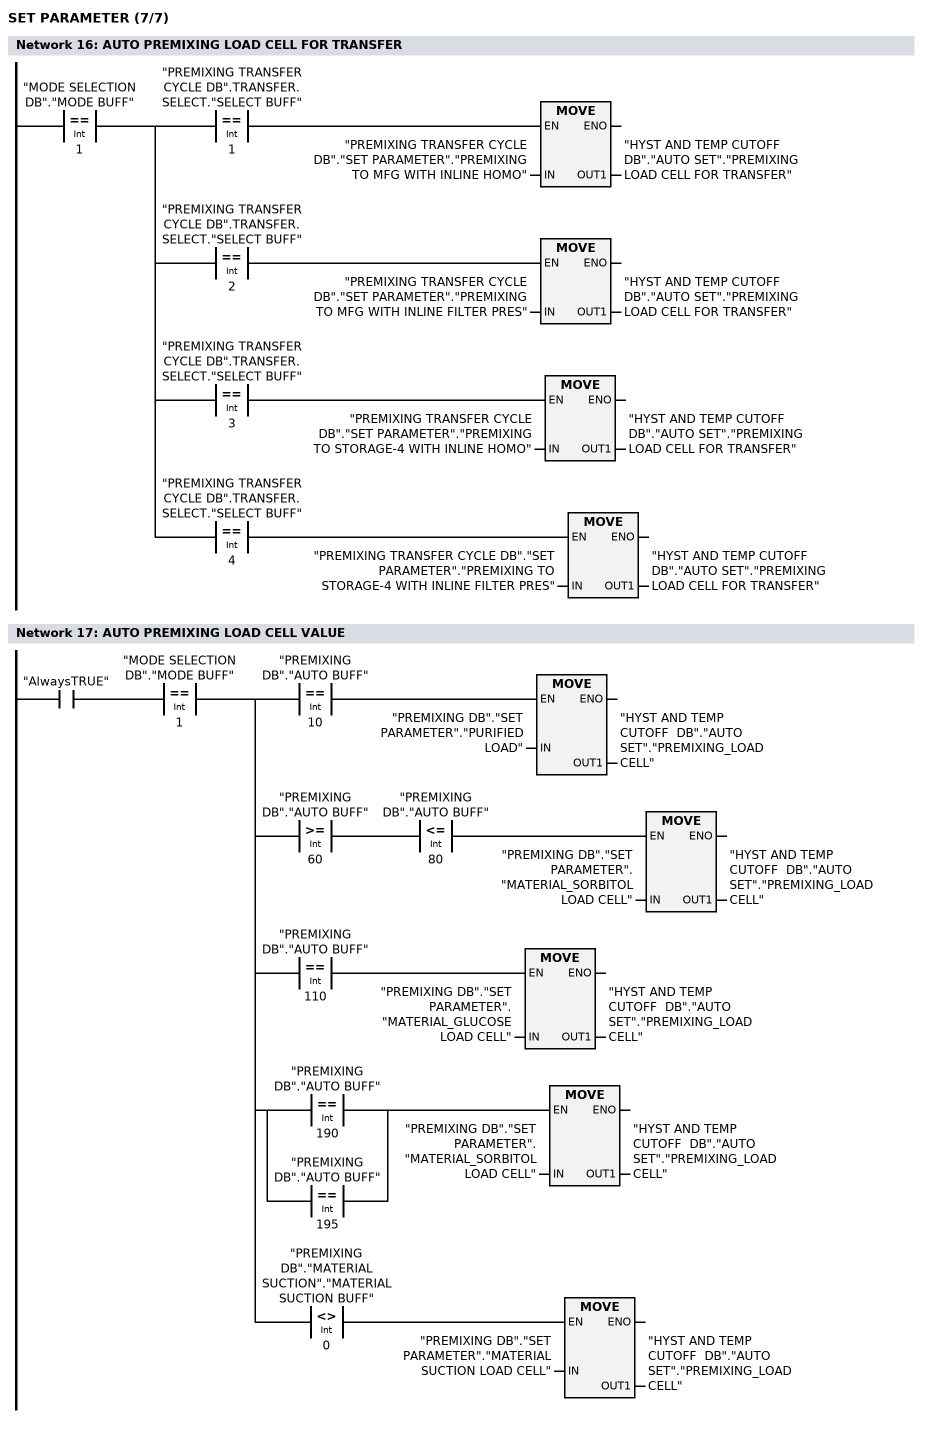
   RUNG wire#powerrail
      { S7_Templates := "SrcType := Int" } EQ_Contact(in1 := "MODE SELECTION DB"."MODE BUFF", in2 := 1)
      wire#w1
      { S7_Templates := "SrcType := Int" } EQ_Contact(in1 := "PREMIXING TRANSFER CYCLE DB".TRANSFER.SELECT."SELECT BUFF", in2 := 1)
      Move(in := "PREMIXING TRANSFER CYCLE DB"."SET PARAMETER"."PREMIXING TO MFG WITH INLINE HOMO", out1 => "HYST AND TEMP CUTOFF  DB"."AUTO SET"."PREMIXING LOAD CELL FOR TRANSFER")
   END_RUNG
   RUNG wire#w1
      { S7_Templates := "SrcType := Int" } EQ_Contact(in1 := "PREMIXING TRANSFER CYCLE DB".TRANSFER.SELECT."SELECT BUFF", in2 := 2)
      Move(in := "PREMIXING TRANSFER CYCLE DB"."SET PARAMETER"."PREMIXING TO MFG WITH INLINE FILTER PRES", out1 => "HYST AND TEMP CUTOFF  DB"."AUTO SET"."PREMIXING LOAD CELL FOR TRANSFER")
   END_RUNG
   RUNG wire#w1
      { S7_Templates := "SrcType := Int" } EQ_Contact(in1 := "PREMIXING TRANSFER CYCLE DB".TRANSFER.SELECT."SELECT BUFF", in2 := 3)
      Move(in := "PREMIXING TRANSFER CYCLE DB"."SET PARAMETER"."PREMIXING TO STORAGE-4 WITH INLINE HOMO", out1 => "HYST AND TEMP CUTOFF  DB"."AUTO SET"."PREMIXING LOAD CELL FOR TRANSFER")
   END_RUNG
   RUNG wire#w1
      { S7_Templates := "SrcType := Int" } EQ_Contact(in1 := "PREMIXING TRANSFER CYCLE DB".TRANSFER.SELECT."SELECT BUFF", in2 := 4)
      Move(in := "PREMIXING TRANSFER CYCLE DB"."SET PARAMETER"."PREMIXING TO STORAGE-4 WITH INLINE FILTER PRES", out1 => "HYST AND TEMP CUTOFF  DB"."AUTO SET"."PREMIXING LOAD CELL FOR TRANSFER")
   END_RUNG
   // the same network as SCL:
   #_w1 := "MODE SELECTION DB"."MODE BUFF" = 1;
   IF #_w1 AND ("PREMIXING TRANSFER CYCLE DB".TRANSFER.SELECT."SELECT BUFF" = 1) THEN
       "HYST AND TEMP CUTOFF  DB"."AUTO SET"."PREMIXING LOAD CELL FOR TRANSFER" := "PREMIXING TRANSFER CYCLE DB"."SET PARAMETER"."PREMIXING TO MFG WITH INLINE HOMO";
   END_IF;
   IF #_w1 AND ("PREMIXING TRANSFER CYCLE DB".TRANSFER.SELECT."SELECT BUFF" = 2) THEN
       "HYST AND TEMP CUTOFF  DB"."AUTO SET"."PREMIXING LOAD CELL FOR TRANSFER" := "PREMIXING TRANSFER CYCLE DB"."SET PARAMETER"."PREMIXING TO MFG WITH INLINE FILTER PRES";
   END_IF;
   IF #_w1 AND ("PREMIXING TRANSFER CYCLE DB".TRANSFER.SELECT."SELECT BUFF" = 3) THEN
       "HYST AND TEMP CUTOFF  DB"."AUTO SET"."PREMIXING LOAD CELL FOR TRANSFER" := "PREMIXING TRANSFER CYCLE DB"."SET PARAMETER"."PREMIXING TO STORAGE-4 WITH INLINE HOMO";
   END_IF;
   IF #_w1 AND ("PREMIXING TRANSFER CYCLE DB".TRANSFER.SELECT."SELECT BUFF" = 4) THEN
       "HYST AND TEMP CUTOFF  DB"."AUTO SET"."PREMIXING LOAD CELL FOR TRANSFER" := "PREMIXING TRANSFER CYCLE DB"."SET PARAMETER"."PREMIXING TO STORAGE-4 WITH INLINE FILTER PRES";
   END_IF;
END_REGION

REGION Network 17: AUTO PREMIXING LOAD CELL VALUE
   RUNG wire#powerrail
      Contact( "AlwaysTRUE" )
      { S7_Templates := "SrcType := Int" } EQ_Contact(in1 := "MODE SELECTION DB"."MODE BUFF", in2 := 1)
      wire#w1
      { S7_Templates := "SrcType := Int" } EQ_Contact(in1 := "PREMIXING DB"."AUTO BUFF", in2 := 10)
      Move(in := "PREMIXING DB"."SET PARAMETER"."PURIFIED LOAD", out1 => "HYST AND TEMP CUTOFF  DB"."AUTO SET"."PREMIXING_LOAD CELL")
   END_RUNG
   RUNG wire#w1
      { S7_Templates := "SrcType := Int" } GE_Contact(in1 := "PREMIXING DB"."AUTO BUFF", in2 := 60)
      { S7_Templates := "SrcType := Int" } LE_Contact(in1 := "PREMIXING DB"."AUTO BUFF", in2 := 80)
      Move(in := "PREMIXING DB"."SET PARAMETER"."MATERIAL_SORBITOL LOAD CELL", out1 => "HYST AND TEMP CUTOFF  DB"."AUTO SET"."PREMIXING_LOAD CELL")
   END_RUNG
   RUNG wire#w1
      { S7_Templates := "SrcType := Int" } EQ_Contact(in1 := "PREMIXING DB"."AUTO BUFF", in2 := 110)
      Move(in := "PREMIXING DB"."SET PARAMETER"."MATERIAL_GLUCOSE LOAD CELL", out1 => "HYST AND TEMP CUTOFF  DB"."AUTO SET"."PREMIXING_LOAD CELL")
   END_RUNG
   RUNG wire#w1
      { S7_Templates := "SrcType := Int" } EQ_Contact(in1 := "PREMIXING DB"."AUTO BUFF", in2 := 190)
      wire#w2
      Move(in := "PREMIXING DB"."SET PARAMETER"."MATERIAL_SORBITOL LOAD CELL", out1 => "HYST AND TEMP CUTOFF  DB"."AUTO SET"."PREMIXING_LOAD CELL")
   END_RUNG
   RUNG wire#w1
      { S7_Templates := "SrcType := Int" } EQ_Contact(in1 := "PREMIXING DB"."AUTO BUFF", in2 := 195)
   END_RUNG wire#w2
   RUNG wire#w1
      { S7_Templates := "SrcType := Int" } NE_Contact(in1 := "PREMIXING DB"."MATERIAL SUCTION"."MATERIAL SUCTION BUFF", in2 := 0)
      Move(in := "PREMIXING DB"."SET PARAMETER"."MATERIAL SUCTION LOAD CELL", out1 => "HYST AND TEMP CUTOFF  DB"."AUTO SET"."PREMIXING_LOAD CELL")
   END_RUNG
   // the same network as SCL:
   #_w1 := "AlwaysTRUE" AND ("MODE SELECTION DB"."MODE BUFF" = 1);
   IF #_w1 AND ("PREMIXING DB"."AUTO BUFF" = 10) THEN
       "HYST AND TEMP CUTOFF  DB"."AUTO SET"."PREMIXING_LOAD CELL" := "PREMIXING DB"."SET PARAMETER"."PURIFIED LOAD";
   END_IF;
   IF #_w1 AND ("PREMIXING DB"."AUTO BUFF" >= 60) AND ("PREMIXING DB"."AUTO BUFF" <= 80) THEN
       "HYST AND TEMP CUTOFF  DB"."AUTO SET"."PREMIXING_LOAD CELL" := "PREMIXING DB"."SET PARAMETER"."MATERIAL_SORBITOL LOAD CELL";
   END_IF;
   IF #_w1 AND ("PREMIXING DB"."AUTO BUFF" = 110) THEN
       "HYST AND TEMP CUTOFF  DB"."AUTO SET"."PREMIXING_LOAD CELL" := "PREMIXING DB"."SET PARAMETER"."MATERIAL_GLUCOSE LOAD CELL";
   END_IF;
   IF #_w1 AND (("PREMIXING DB"."AUTO BUFF" = 190) OR ("PREMIXING DB"."AUTO BUFF" = 195)) THEN
       "HYST AND TEMP CUTOFF  DB"."AUTO SET"."PREMIXING_LOAD CELL" := "PREMIXING DB"."SET PARAMETER"."MATERIAL_SORBITOL LOAD CELL";
   END_IF;
   IF #_w1 AND ("PREMIXING DB"."MATERIAL SUCTION"."MATERIAL SUCTION BUFF" <> 0) THEN
       "HYST AND TEMP CUTOFF  DB"."AUTO SET"."PREMIXING_LOAD CELL" := "PREMIXING DB"."SET PARAMETER"."MATERIAL SUCTION LOAD CELL";
   END_IF;
END_REGION
END_FUNCTION
